PROGRAM PRG_3_PMPS_POST
VAR
    fbArbiterIO: FB_SubSysToArbiter_IO;
    fb_vetoArbiter: FB_VetoArbiter;

    bST3K4_Veto: BOOL;
    bM1K1Veto: BOOL;
    bST4K4_Veto:BOOL;
END_VAR

bST3K4_Veto := PMPS_GVL.stCurrentBeamParameters.aVetoDevices[PMPS.K_Stopper.ST3K4];
bST4K4_Veto := PMPS_GVL.stCurrentBeamParameters.aVetoDevices[PMPS.K_Stopper.ST4K4];
bM1K1Veto := NOT PMPS_GVL.stCurrentBeamParameters.aVetoDevices[PMPS.K_Stopper.MR1K1_OUT]
                AND PMPS_GVL.stCurrentBeamParameters.aVetoDevices[PMPS.K_Stopper.MR1K1_IN];

fbArbiterIO(
    i_bVeto:=bST3K4_Veto,
    Arbiter:=fbArbiter,
    fbFFHWO:=fbFastFaultOutput1);

fb_vetoArbiter(bVeto:=bST4K4_Veto OR bST3K4_Veto OR bM1K1Veto,
                HigherAuthority := GVL_PMPS.fbArbiter,
                LowerAuthority := GVL_PMPS.fbArbiter2,
                FFO := GVL_PMPS.fbFastFaultOutput2);

fbFastFaultOutput1.Execute(i_xVeto:=bST3K4_Veto OR bM1K1Veto);
fbFastFaultOutput2.Execute(i_xVeto:=bST3K4_Veto OR bM1K1Veto OR bST4K4_Veto); // Eventually, also veto on ST4K4 using OR

END_PROGRAM

(* stored: Version 1.1.0.1, ProductVersion 3.1.4022.18
   POU PRG_3_PMPS_POST: Id {ec0299d5-08dd-4c37-8c55-47b9e81fd84b}, SpecialFunc None *)
